// TIA Portal project "PLCII_Pro2" (V15.1)

(* hardware
DEVICE "S7-1200 station_1"  S7-1200 Station
   slot 0: "Rack_0"  S7-1200 Rack  Rack  V1.0
   slot 1: "PLC_1"  CPU 1215C DC/DC/Rly  6ES7 215-1HG40-0XB0  V4.2
*)

// ===== PLC "PLC_1"  CPU 1215C DC/DC/Rly =====

VAR_GLOBAL   // PLC tag table "Default tag table"
   "Start" AT %M0.0 : Bool;
   "Sys_runing" AT %M0.1 : Bool;
   "Stop" AT %M0.2 : Bool;
   "Activate" AT %M0.3 : Bool;
   "Sys_Activated" AT %M0.4 : Bool;
END_VAR

DATA_BLOCK "DigitalFilingSys_DB"   // DB1
{ S7_Optimized_Access := 'TRUE' }
VERSION : 0.1
// stored: InstanceOfName DigitalFilingSys
"DigitalFilingSys"
BEGIN
END_DATA_BLOCK

DATA_BLOCK "System_DB"   // DB2
{ S7_Optimized_Access := 'TRUE' }
VERSION : 0.1
   VAR
      ProxSW : Bool;
      LevelSW : Bool;
      RedPE : Bool;
      BluePE : Bool;
      BoxState : Int;
      ConvoyerMotor_State : Int;
      WalnutHopper : Bool;
      PecanHopper : Bool;
      Motor : Bool;
   END_VAR
BEGIN
END_DATA_BLOCK

FUNCTION_BLOCK "DigitalFilingSys"   // FB1, LAD
{ S7_Optimized_Access := 'TRUE' }
VERSION : 0.1
   VAR
      ONS1 : Bool;
      ONS2 : Bool;
      ONS3 : Bool;
   END_VAR
   VAR_TEMP   // added for the SCL form of the ladder/FBD networks
      _w1 : Bool;
      _w2 : Bool;
      _w3 : Bool;
      _w4 : Bool;
      _w5 : Bool;
   END_VAR
BEGIN

REGION Network 1: Start-up
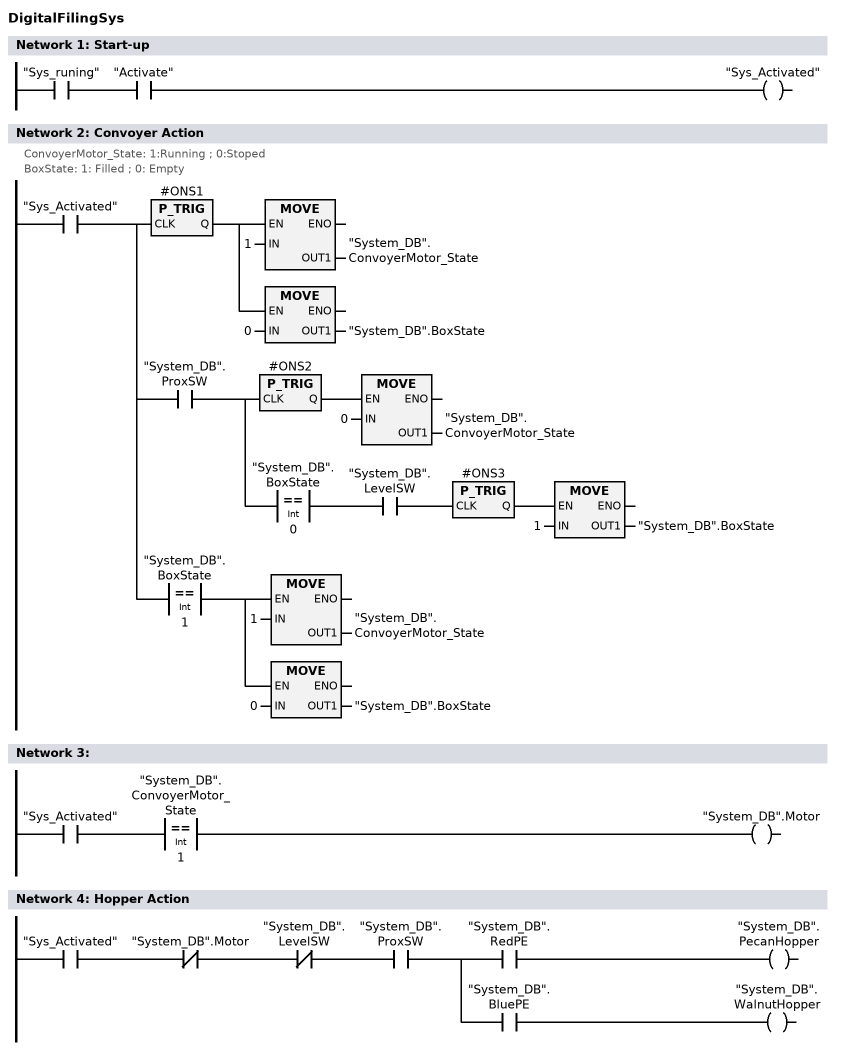
   RUNG wire#powerrail
      Contact( "Sys_runing" )
      Contact( "Activate" )
      Coil( "Sys_Activated" )
   END_RUNG
   // the same network as SCL:
   "Sys_Activated" := "Sys_runing" AND "Activate";
END_REGION

REGION Network 2: Convoyer Action
   // ConvoyerMotor_State: 1:Running ; 0:Stoped
   // BoxState: 1: Filled ; 0: Empty
   RUNG wire#powerrail
      Contact( "Sys_Activated" )
      wire#w1
      P_Trig( #ONS1 )
      wire#w2
      Move(in := 1, out1 => "System_DB".ConvoyerMotor_State)
   END_RUNG
   RUNG wire#w2
      Move(in := 0, out1 => "System_DB".BoxState)
   END_RUNG
   RUNG wire#w1
      Contact( "System_DB".ProxSW )
      wire#w3
      P_Trig( #ONS2 )
      Move(in := 0, out1 => "System_DB".ConvoyerMotor_State)
   END_RUNG
   RUNG wire#w3
      { S7_Templates := "SrcType := Int" } EQ_Contact(in1 := "System_DB".BoxState, in2 := 0)
      Contact( "System_DB".LevelSW )
      P_Trig( #ONS3 )
      Move(in := 1, out1 => "System_DB".BoxState)
   END_RUNG
   RUNG wire#w1
      { S7_Templates := "SrcType := Int" } EQ_Contact(in1 := "System_DB".BoxState, in2 := 1)
      wire#w4
      Move(in := 1, out1 => "System_DB".ConvoyerMotor_State)
   END_RUNG
   RUNG wire#w4
      Move(in := 0, out1 => "System_DB".BoxState)
   END_RUNG
   // the same network as SCL:
   #_w1 := "Sys_Activated" AND NOT #ONS1;   // rising edge
   #ONS1 := "Sys_Activated";
   IF #_w1 THEN
       "System_DB".ConvoyerMotor_State := 1;
       "System_DB".BoxState := 0;
   END_IF;
   #_w2 := "Sys_Activated" AND "System_DB".ProxSW;
   #_w3 := #_w2 AND NOT #ONS2;   // rising edge
   #ONS2 := #_w2;
   IF #_w3 THEN "System_DB".ConvoyerMotor_State := 0; END_IF;
   #_w4 := #_w2 AND ("System_DB".BoxState = 0) AND "System_DB".LevelSW;
   #_w5 := #_w4 AND NOT #ONS3;   // rising edge
   #ONS3 := #_w4;
   IF #_w5 THEN "System_DB".BoxState := 1; END_IF;
   IF "Sys_Activated" AND ("System_DB".BoxState = 1) THEN
       "System_DB".ConvoyerMotor_State := 1;
       "System_DB".BoxState := 0;
   END_IF;
END_REGION

REGION Network 3
   RUNG wire#powerrail
      Contact( "Sys_Activated" )
      { S7_Templates := "SrcType := Int" } EQ_Contact(in1 := "System_DB".ConvoyerMotor_State, in2 := 1)
      Coil( "System_DB".Motor )
   END_RUNG
   // the same network as SCL:
   "System_DB".Motor := "Sys_Activated" AND ("System_DB".ConvoyerMotor_State = 1);
END_REGION

REGION Network 4: Hopper Action
   RUNG wire#powerrail
      Contact( "Sys_Activated" )
      I_Contact( "System_DB".Motor )
      I_Contact( "System_DB".LevelSW )
      Contact( "System_DB".ProxSW )
      wire#w1
      Contact( "System_DB".RedPE )
      Coil( "System_DB".PecanHopper )
   END_RUNG
   RUNG wire#w1
      Contact( "System_DB".BluePE )
      Coil( "System_DB".WalnutHopper )
   END_RUNG
   // the same network as SCL:
   #_w1 := "Sys_Activated" AND NOT "System_DB".Motor AND NOT "System_DB".LevelSW AND "System_DB".ProxSW;
   "System_DB".PecanHopper := #_w1 AND "System_DB".RedPE;
   "System_DB".WalnutHopper := #_w1 AND "System_DB".BluePE;
END_REGION
END_FUNCTION_BLOCK

FUNCTION "Hopper" : Void   // FC1, FBD
{ S7_Optimized_Access := 'TRUE' }
VERSION : 0.1
   VAR_INPUT
      ColorSw : Bool;
   END_VAR
   VAR_OUTPUT
      HopperColor : Bool;
   END_VAR
BEGIN

REGION Network 1
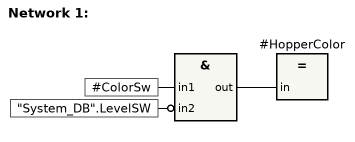
   #HopperColor := #ColorSw AND NOT "System_DB".LevelSW;
END_REGION
END_FUNCTION

ORGANIZATION_BLOCK "Main"   // OB1, LAD, ProgramCycle
TITLE = "Main Program Sweep (Cycle)"
{ S7_Optimized_Access := 'TRUE' }
VERSION : 0.1
   VAR_INPUT
      Initial_Call : Bool;   // Initial call of this OB
      Remanence : Bool;   // =True, if remanent data are available
   END_VAR
BEGIN

REGION Network 1
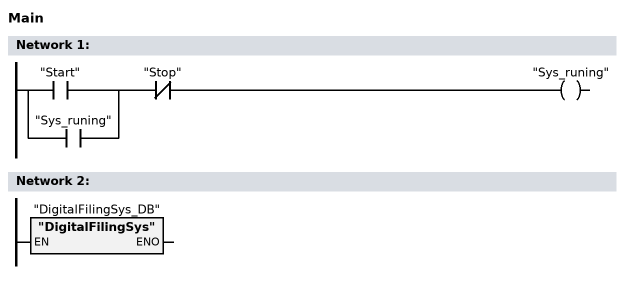
   RUNG wire#powerrail
      Contact( "Start" )
      wire#w1
      I_Contact( "Stop" )
      Coil( "Sys_runing" )
   END_RUNG
   RUNG wire#powerrail
      Contact( "Sys_runing" )
   END_RUNG wire#w1
   // the same network as SCL:
   "Sys_runing" := ("Start" OR "Sys_runing") AND NOT "Stop";
END_REGION

REGION Network 2
   RUNG wire#powerrail
      "DigitalFilingSys_DB"()
   END_RUNG
   // the same network as SCL:
   "DigitalFilingSys_DB"();   // "DigitalFilingSys"
END_REGION
END_ORGANIZATION_BLOCK